(* Logix 5000 project; controller Robot_Index_Table Emulate 5570 rev 33.11; software revision 33.00 *)

TASK MainTask (continuous, watchdog 500 ms) : MainProgram, EMULATION

MODULES
   Local : Emulate 5570 (ICP 2, rev 33.11)
       : 1756-IB16 (ICP 3, rev 3.1, Input RPI 20 ms)
       : vendor 1 type 7 code 16 (ICP 4, rev 3.1, Output RPI 20 ms)
END_MODULES

PROGRAM EMULATION   (* main routine EMULATION *)
VAR
   COUNTER0 : COUNTER := (PRE := 3);
   ONS1 : BOOL;
   TIMER0 : TIMER := (PRE := 4000);
   TIMER1 : TIMER := (PRE := 1200);
   TIMER2 : TIMER := (PRE := 3000);
   TIMER3 : TIMER := (PRE := 4000);
   TIMER4 : TIMER := (PRE := 2000);
END_VAR

ROUTINE EMULATION   (* ladder *)
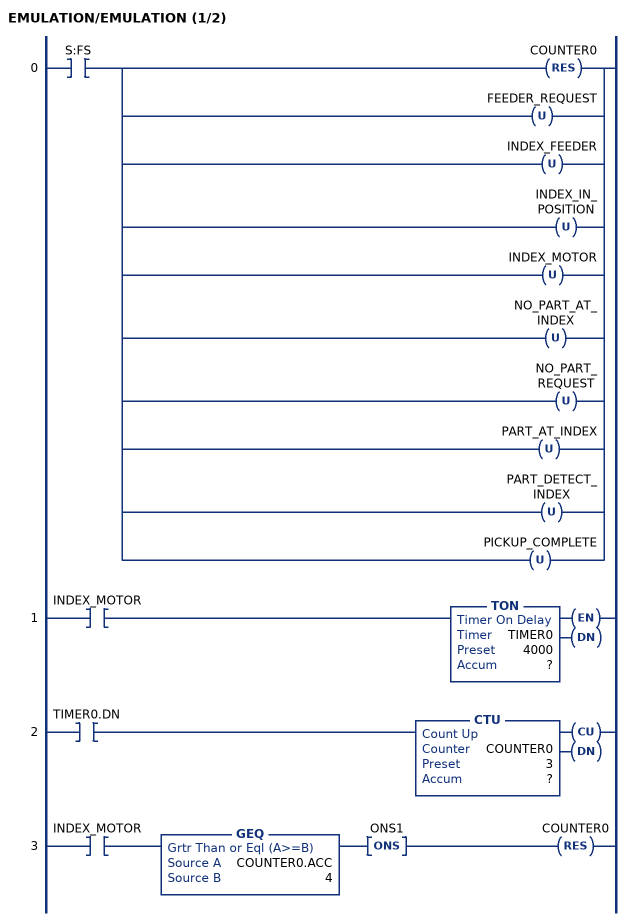
   0: XIC(S:FS)[RES(COUNTER0) ,OTU(FEEDER_REQUEST) ,OTU(INDEX_FEEDER) ,OTU(INDEX_IN_POSITION) ,OTU(INDEX_MOTOR) ,OTU(NO_PART_AT_INDEX) ,OTU(NO_PART_REQUEST) ,OTU(PART_AT_INDEX) ,OTU(PART_DETECT_INDEX) ,OTU(PICKUP_COMPLETE) ];
   1: XIC(INDEX_MOTOR)TON(TIMER0,?,?);
   2: XIC(TIMER0.DN)CTU(COUNTER0,?,?);
   3: XIC(INDEX_MOTOR)GEQ(COUNTER0.ACC,4)ONS(ONS1)RES(COUNTER0);
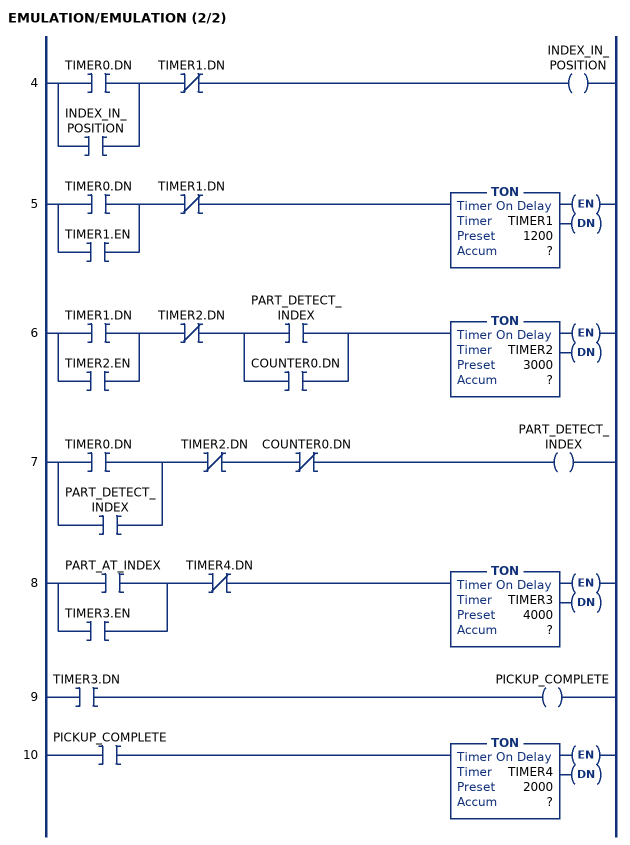
   4: [XIC(TIMER0.DN) ,XIC(INDEX_IN_POSITION) ]XIO(TIMER1.DN)OTE(INDEX_IN_POSITION);
   5: [XIC(TIMER0.DN) ,XIC(TIMER1.EN) ]XIO(TIMER1.DN)TON(TIMER1,?,?);
   6: [XIC(TIMER1.DN) ,XIC(TIMER2.EN) ]XIO(TIMER2.DN)[XIC(PART_DETECT_INDEX) ,XIC(COUNTER0.DN) ]TON(TIMER2,?,?);
   7: [XIC(TIMER0.DN) ,XIC(PART_DETECT_INDEX) ]XIO(TIMER2.DN)XIO(COUNTER0.DN)OTE(PART_DETECT_INDEX);
   8: [XIC(PART_AT_INDEX) ,XIC(TIMER3.EN) ]XIO(TIMER4.DN)TON(TIMER3,?,?);
   9: XIC(TIMER3.DN)OTE(PICKUP_COMPLETE);
   10: XIC(PICKUP_COMPLETE)TON(TIMER4,?,?);
END_ROUTINE
END_PROGRAM

PROGRAM MainProgram   (* main routine MainRoutine *)

ROUTINE MainRoutine   (* ladder *)
   0: ;
END_ROUTINE
END_PROGRAM
